# EPICS autosave request: apps/agilentApp/Db/A6551_settings.req
$(P):imon.HIHI
$(P):imon.LOLO
$(P):imon.HIGH
$(P):imon.LOW
$(P):imon.HSV
$(P):imon.HHSV
$(P):imon.LSV
$(P):imon.LLSV
$(P):vmon.HIHI
$(P):vmon.LOLO
$(P):vmon.HIGH
$(P):vmon.LOW
$(P):vmon.HSV
$(P):vmon.HHSV
$(P):vmon.LSV
$(P):vmon.LLSV
$(P):vset.DRVH
$(P):iset.DRVH
